TYPE ST_Machine_Cmd :
	STRUCT
		MoveAll : BOOL;
	END_STRUCT
END_TYPE

(* stored: Version 1.1.0.1
   DUT ST_Machine_Cmd: Id {a947bc9e-ed7c-477f-adfc-e81c741493a1} *)
